FUNCTION_BLOCK conv2_wkpc_colorsense (* A simple FB with a single algorithm and REQ/CNF pair *)
  (* Standard: 61499-1 *)
  (* Version 0.0, 2006-09-03, JHC, Holobloc Inc *)
  (* Compiler header: package fb.rt.template; *)
  (* Compiler classdef: SimpleFB *)
  (* Compiler Java Sun JDK 1.5.0 *)
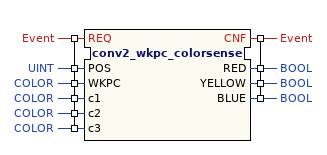
  EVENT_INPUT
    REQ WITH POS, WKPC, c1, c2, c3; (* Normal Execution Request *)
  END_EVENT
  EVENT_OUTPUT
    CNF WITH RED, YELLOW, BLUE; (* Execution Confirmation *)
  END_EVENT
  VAR_INPUT
    POS : UINT;
    WKPC : COLOR;
    c1 : COLOR;
    c2 : COLOR;
    c3 : COLOR;
  END_VAR
  VAR_OUTPUT
    RED : BOOL;
    YELLOW : BOOL;
    BLUE : BOOL;
  END_VAR
  ALGORITHM REQ IN ST: (* Normally executed algorithm *)
IF POS = 50 AND WKPC = c1 THEN
RED := TRUE;
ELSIF POS = 75 AND WKPC = c2 THEN
YELLOW := TRUE;
ELSIF POS = 100 AND WKPC = c3 THEN
BLUE := TRUE;
ELSE
RED := FALSE;
YELLOW := FALSE;
BLUE := FALSE;
END_IF;
  END_ALGORITHM
END_FUNCTION_BLOCK
